IF nPlayerOne = 0 AND  nPlayerTwo = 0 THEN
	sWinner := '';
	xPlayerOneWins := FALSE;
	xPlayerTwoWins := FALSE;
END_IF

FOR i := 5 TO 49 DO //Set to 5 so as not to overwrite staff names

	IF 	CurrentMonthSignInTable[i].Name = '' THEN
	sPlayerList[i] := CurrentMonthSignInTable[i-5].Name;
	ELSE
	EXIT;	
	END_IF

END_FOR

ACTION Play11s:

END_ACTION

ACTION Play5s:

END_ACTION

END_PROGRAM

// ---- HMI/VariableHandleForHmi.TcPOU
PROGRAM VariableHandleForHmi
VAR
END_VAR

numberOfOpenWindows := EnOcean.totalNumberOfWindowsOpen;
boardroomModeIsProjector := LightControl.xBoardRoom_Lights_ProjectorMode;
boardroomModeIsFullOn := PTM200StrippedTables[3].Signal OR PTM200StrippedTables[2].Signal;
communalOccupancy1 := Dali.CommunalAreaPIR_1_Occupancy;
communalOccupancy2 := Dali.CommunalAreaPIR_2_Occupancy;
staffOccupancy1 := Dali.StaffroomPIR_1_Occupancy;
staffOccupancy2 := Dali.StaffroomPIR_2_Occupancy;
boardOccupancy1 := Dali.BoardroomPIR_1_Occupancy;
boardOccupancy2 := Dali.BoardroomPIR_2_Occupancy;
communalLux1 := Dali.CommunalAreaPIR_1_LuxLevel;
communalLux2 := Dali.CommunalAreaPIR_2_LuxLevel;
staffLux1 := Dali.StaffroomPIR_1_LuxLevel;
staffLux2 := Dali.StaffroomPIR_2_LuxLevel;
boardLux1 := Dali.BoardroomPIR_1_LuxLevel;
boardLux2 := Dali.BoardroomPIR_2_LuxLevel;

END_PROGRAM

// ---- WORKSHOP WALL/PowerSupply.TcPOU
PROGRAM PowerSupply
VAR
	triggerCoeRead							:	Pulse;
	readPsuDiagData							:	FB_EcCoESdoReadEx;
	readPsuInfoData							:	FB_EcCoESdoReadEx;
	psuDiagData								:	ST_PsuDiagData;
	psuInfoData								:	ST_PsuInfoData;
	testArr									:	ARRAY [1..20] OF BYTE;
	amsAdr							AT%I*	:	ST_AmsAddr;
	psuWarning						AT%I*	:	BOOL;
	psuError						AT%I*	:	BOOL;
	psuDcOk							AT%I*	:	BOOL;
	psuOutVoltage					AT%I*	:	REAL;
	psuOutCurrent					AT%I*	:	REAL;
	psuInputUnderVoltage			AT%I*	:	BOOL;
	psuDisableOutput				AT%Q*	:	BOOL;
END_VAR

triggerCoeRead(enable:= TRUE, offTime:= T#0.5S, onTime:= T#0.5S, Q=> );

readPsuDiagData(
	sNetId:= F_CreateAmsNetId(amsAdr.netId), 
	nSlaveAddr:= amsAdr.port, 
	nSubIndex:= 16#01, 
	nIndex:= 16#FA14, 
	pDstBuf:= ADR(psuDiagData), 
	cbBufLen:= SIZEOF(psuDiagData), 
	bExecute:= triggerCoeRead.Q, 
	tTimeout:= , 
	bCompleteAccess:= TRUE, 
	bBusy=> , 
	bError=> , 
	nErrId=> , 
	cbRead=> );
	
readPsuInfoData(
	sNetId:= F_CreateAmsNetId(amsAdr.netId), 
	nSlaveAddr:= amsAdr.port, 
	nSubIndex:= 16#01, 
	nIndex:= 16#F914, 
	pDstBuf:= ADR(psuInfoData), 
	cbBufLen:= SIZEOF(psuInfoData), 
	bExecute:= triggerCoeRead.Q, 
	tTimeout:= , 
	bCompleteAccess:= TRUE, 
	bBusy=> , 
	bError=> , 
	nErrId=> , 
	cbRead=> );

END_PROGRAM

// ---- BLINDS/ConvertBoolArrayToString.TcPOU
FUNCTION_BLOCK ConvertBoolArrayToString
VAR_INPUT
	boolArray: ARRAY[1..16] OF BOOL;
END_VAR
VAR_OUTPUT
	resultString: STRING := '';
END_VAR
VAR
	i: INT := 1;
END_VAR

FOR i := 1 TO 15 by 1 DO
    IF boolArray[i] THEN
        resultString := Concat(STR1 := resultString, STR2 := '1');
    ELSE
        resultString := Concat(STR1 := resultString, STR2 := '0');
    END_IF;
END_FOR;

END_FUNCTION_BLOCK

// ---- BLINDS/fConvertBoolArrayToString.TcPOU
FUNCTION fConvertBoolArrayToString : STRING
VAR_INPUT
	boolArray: ARRAY[1..16] OF BOOL;
END_VAR
VAR
	i: INT := 1;
END_VAR

FOR i := 1 TO 16 BY 1 DO
    IF boolArray[i] THEN
        fConvertBoolArrayToString := Concat(STR1 := fConvertBoolArrayToString, STR2 := '1');
    ELSE
        fConvertBoolArrayToString := Concat(STR1 := fConvertBoolArrayToString, STR2 := '0');
    END_IF;
END_FOR;

END_FUNCTION

// ---- BLINDS/PrgMqttCom_Blinds_Publisher.TcPOU
PROGRAM PrgMqttCom_Blinds_Publisher
VAR
	fbMqttClient : FB_IotMqttClient;
	bSetParameter : BOOL := TRUE;
	bConnect : BOOL := TRUE;
	
	(* published message *)
	sTopicSelectRoom : STRING(255);//:= 'Staff Room';
	sTopicSelectBulkCommand : STRING(255) := 'Blind Selection';
	//sTopicSelectBoardroom : STRING(255) := 'Boardroom';
	
	bSelectStaffRoom : BOOL;
	bSelectCommunalArea : BOOL;
	bSelectBoardroom : BOOL;
	
	sPayloadCommand : STRING(255);// := 'Up';
//	sPayloadCommandDown : STRING(255) := 'Down';
//	sPayloadCommandStop : STRING(255) := 'Stop';
//	sPayloadCommandTilt : STRING(255) := 'Tilt';

	bCommandUp : BOOL;
	bCommandDown : BOOL;
	bCommandStop : BOOL;
	bCommandTilt : BOOL;
	
	bulkCommandPackage :STRING;
	
	i: INT;
	fbTimer : TON := (PT:=T#1S);
	fbTimerTilt : TON := (PT:=T#0.5S);
	
	fbMessageQueue : FB_IotMqttMessageQueue;
	fbMessage : FB_IotMqttMessage;
	
	hrErrorOccurred : HRESULT; // contains the latest occurred error
END_VAR

IF bSetParameter THEN
	bSetParameter := FALSE;
	fbMqttClient.sHostName:= '10.199.143.2';
	fbMqttClient.nHostPort:= 1883;
	fbMqttClient.sClientId:= 'CX2040_Blinds'; 
	fbMqttClient.sTopicPrefix:= ''; 
	fbMqttClient.nKeepAlive:= 60; 
//	fbMqttClient.sUserName:= ;
//	fbMqttClient.sUserPassword:= ; 
//	fbMqttClient.stWill:= ; 
//	fbMqttClient.stTLS:= ;
	fbMqttClient.ipMessageQueue := fbMessageQueue;
END_IF

fbMqttClient.Execute(bConnect);
IF fbMqttClient.bError THEN
	// add your error logging here
	hrErrorOccurred := fbMqttClient.hrErrorCode;
END_IF

IF bSelectStaffRoom THEN
	bSelectStaffRoom := FALSE;
	sTopicSelectRoom := 'Staff Room';
	bulkCommandPackage := fConvertBoolArrayToString(boolArray := BackgroundComms.BlindCommandTable[0].SelectBlindsBulkCommand);
END_IF

IF bSelectCommunalArea THEN
	bSelectCommunalArea := FALSE;
	sTopicSelectRoom := 'Communal Area';
	bulkCommandPackage := fConvertBoolArrayToString(boolArray := BackgroundComms.BlindCommandTable[1].SelectBlindsBulkCommand);
END_IF

IF bSelectBoardroom THEN
	bSelectBoardroom := FALSE;
	sTopicSelectRoom := 'Boardroom';
	bulkCommandPackage := fConvertBoolArrayToString(boolArray := BackgroundComms.BlindCommandTable[2].SelectBlindsBulkCommand);
END_IF



IF bCommandUp THEN
	bCommandUp := FALSE;
	sPayloadCommand := 'Up';
	IF sTopicSelectRoom = 'Staff Room' THEN
		bSelectStaffRoom := TRUE;
	ELSIF sTopicSelectRoom = 'Communal Area' THEN
		bulkCommandPackage := fConvertBoolArrayToString(boolArray := BackgroundComms.BlindCommandTable[1].SelectBlindsBulkCommand);
	ELSIF sTopicSelectRoom = 'Boardroom' THEN
		bulkCommandPackage := fConvertBoolArrayToString(boolArray := BackgroundComms.BlindCommandTable[2].SelectBlindsBulkCommand);
	END_IF
END_IF

IF bCommandDown THEN
	bCommandDown := FALSE;
	sPayloadCommand := 'Down';
	IF sTopicSelectRoom = 'Staff Room' THEN
		bSelectStaffRoom := TRUE;//bulkCommandPackage := fConvertBoolArrayToString(boolArray := BackgroundComms.BlindCommandTable[0].SelectBlindsBulkCommand);
	ELSIF sTopicSelectRoom = 'Communal Area' THEN
		bulkCommandPackage := fConvertBoolArrayToString(boolArray := BackgroundComms.BlindCommandTable[1].SelectBlindsBulkCommand);
	ELSIF sTopicSelectRoom = 'Boardroom' THEN
		bulkCommandPackage := fConvertBoolArrayToString(boolArray := BackgroundComms.BlindCommandTable[2].SelectBlindsBulkCommand);
	END_IF
END_IF

IF bCommandStop THEN
	bCommandStop := FALSE;
	sPayloadCommand := 'Stop';
	IF sTopicSelectRoom = 'Staff Room' THEN
		bSelectStaffRoom := TRUE;//bulkCommandPackage := fConvertBoolArrayToString(boolArray := BackgroundComms.BlindCommandTable[0].SelectBlindsBulkCommand);
	ELSIF sTopicSelectRoom = 'Communal Area' THEN
		bulkCommandPackage := fConvertBoolArrayToString(boolArray := BackgroundComms.BlindCommandTable[1].SelectBlindsBulkCommand);
	ELSIF sTopicSelectRoom = 'Boardroom' THEN
		bulkCommandPackage := fConvertBoolArrayToString(boolArray := BackgroundComms.BlindCommandTable[2].SelectBlindsBulkCommand);
	END_IF
END_IF

IF bCommandTilt THEN
	bCommandTilt := FALSE;
	sPayloadCommand := 'Tilt';
	IF sTopicSelectRoom = 'Staff Room' THEN
		bSelectStaffRoom := TRUE;//bulkCommandPackage := fConvertBoolArrayToString(boolArray := BackgroundComms.BlindCommandTable[0].SelectBlindsBulkCommand);
	ELSIF sTopicSelectRoom = 'Communal Area' THEN
		bulkCommandPackage := fConvertBoolArrayToString(boolArray := BackgroundComms.BlindCommandTable[1].SelectBlindsBulkCommand);
	ELSIF sTopicSelectRoom = 'Boardroom' THEN
		bulkCommandPackage := fConvertBoolArrayToString(boolArray := BackgroundComms.BlindCommandTable[2].SelectBlindsBulkCommand);
	END_IF
END_IF





IF fbMqttClient.bConnected THEN
	IF sPayloadCommand = 'Tilt' THEN
		fbTimerTilt(IN:=TRUE);
		fbMqttClient.Publish(	sTopic:= sTopicSelectBulkCommand, 
									pPayload:= ADR(bulkCommandPackage), nPayloadSize:= LEN2(ADR(bulkCommandPackage))+1, 
									eQoS:= TcIotMqttQos.AtMostOnceDelivery, bRetain:= FALSE, bQueue:= FALSE );
		fbMqttClient.Publish(	sTopic:= sTopicSelectRoom, 
									pPayload:= ADR(sPayloadCommand), nPayloadSize:= LEN2(ADR(sPayloadCommand))+1, 
									eQoS:= TcIotMqttQos.AtMostOnceDelivery, bRetain:= FALSE, bQueue:= FALSE );
		
		IF fbTimerTilt.Q THEN // publish new payload every second
			sPayloadCommand := 'Stop';
			fbTimerTilt(IN:=FALSE);
			fbMqttClient.Publish(	sTopic:= sTopicSelectBulkCommand, 
									pPayload:= ADR(bulkCommandPackage), nPayloadSize:= LEN2(ADR(bulkCommandPackage))+1, 
									eQoS:= TcIotMqttQos.AtMostOnceDelivery, bRetain:= FALSE, bQueue:= FALSE );
			fbMqttClient.Publish(	sTopic:= sTopicSelectRoom, 
									pPayload:= ADR(sPayloadCommand), nPayloadSize:= LEN2(ADR(sPayloadCommand))+1, 
									eQoS:= TcIotMqttQos.AtMostOnceDelivery, bRetain:= FALSE, bQueue:= FALSE );			
			IF fbMqttClient.bError THEN
				// add your error logging here
				hrErrorOccurred := fbMqttClient.hrErrorCode;
			END_IF
		END_IF
	ELSE
		fbTimer(IN:=TRUE);
		IF fbTimer.Q THEN // publish new payload every second
			fbTimer(IN:=FALSE);
			fbMqttClient.Publish(	sTopic:= sTopicSelectBulkCommand, 
									pPayload:= ADR(bulkCommandPackage), nPayloadSize:= LEN2(ADR(bulkCommandPackage))+1, 
									eQoS:= TcIotMqttQos.AtMostOnceDelivery, bRetain:= FALSE, bQueue:= FALSE );
									
			fbMqttClient.Publish(	sTopic:= sTopicSelectRoom, 
									pPayload:= ADR(sPayloadCommand), nPayloadSize:= LEN2(ADR(sPayloadCommand))+1, 
									eQoS:= TcIotMqttQos.AtMostOnceDelivery, bRetain:= FALSE, bQueue:= FALSE );
			IF fbMqttClient.bError THEN
				// add your error logging here
				hrErrorOccurred := fbMqttClient.hrErrorCode;
			END_IF
		END_IF
	END_IF
END_IF

fbTimerTilt();

END_PROGRAM

// ---- HMI/ReadCP67.TcPOU
PROGRAM ReadCP67
VAR
	
	ReadActLightLvlBoardroom :FB_DALIV2QueryActualLevel;  //Used to read back actual light lvl to correct dimmer on CP67 ask Plug top


	ADS_READ:ADSREAD;
	
	ADX_READ_DMXR:ADSREAD;
	ADX_READ_DMXG:ADSREAD;
	ADX_READ_DMXB:ADSREAD;
	
	DMX_Enable_READ:ADSREAD;
	
	HoldCP67BoardRoomLightsOn:BYTE;
	

	Sample		: BYTE;
	
	DMXRValues	:	ARRAY [0..7] OF BYTE;
	DMXGValues	:	ARRAY [0..7] OF BYTE;
	DMXBValues	:	ARRAY [0..7] OF BYTE;
	
	CP67_DMX_Enable	:	BOOL;
	
	FBDALIV2Dimmer1Switch : ARRAY [1..15] OF FB_DALIV2Dimmer1Switch;
	CASECP67BoardRoomLightsOn : INT;

END_VAR

sample := sample + 1;

FBDALIV2Dimmer1Switch[1](stCommandBuffer:= stCommandBuffer);
FBDALIV2Dimmer1Switch[2](stCommandBuffer:= stCommandBuffer);
ReadActLightLvlBoardroom(stCommandBuffer := stCommandBuffer , nActualLevel => BoardroomActualLightLvl ); 

IF CP67BoardRoomLightsOn <> HoldCP67BoardRoomLightsOn THEN
HoldCP67BoardRoomLightsOn := CP67BoardRoomLightsOn;
CASECP67BoardRoomLightsOn := 10;
END_IF

	CASE CASECP67BoardRoomLightsOn OF
		
	0: //Idle
	
	10:	FBDALIV2Dimmer1Switch[1].nDimmValue	:=  CP67BoardRoomLightsOn;
		FBDALIV2Dimmer1Switch[1].nAddr		:= 3;
		FBDALIV2Dimmer1Switch[1].eAddrType	:= 1;
			
		FBDALIV2Dimmer1Switch[2].nDimmValue	:=  CP67BoardRoomLightsOn; 
		FBDALIV2Dimmer1Switch[2].nAddr		:= 2; 
		FBDALIV2Dimmer1Switch[2].eAddrType	:= 1;
			
		CASECP67BoardRoomLightsOn			:= 20;	
			
	20:	IF  NOT FBDALIV2Dimmer1Switch[1].bBusy AND NOT FBDALIV2Dimmer1Switch[2].bBusy THEN
		CASECP67BoardRoomLightsOn 			:= 30;	

		ReadActLightLvlBoardroom.bStart		:= TRUE;
		ReadActLightLvlBoardroom.nAddr		:= 6;
		ReadActLightLvlBoardroom.eAddrType	:= 0;
		END_IF
	
	30:	IF NOT ReadActLightLvlBoardroom.bBusy THEN
		ReadActLightLvlBoardroom.bStart			:= FALSE;
		CASECP67BoardRoomLightsOn 				:= 0;
		
		END_IF
				
		
	END_CASE
		
	
	
	
(*// Send back actual light lvls for slider on CP67	
ReadActLightLvlBoardroom(
	bStart:= Sample.0, 
	nAddr:= 6, 
	eAddrType:= 0, 
	eCommandPriority:= , 
	bBusy=> , 
	bError=> , 
	nErrorId=> , 
	nActualLevel=> BoardroomActualLightLvl, 
	stCommandBuffer:= stCommandBuffer);	*)

(*
// DMX Values	
ADX_READ_DMXR(
	NETID:= '192.168.3.8.1.1', 
	PORT:= 851, 
	IDXGRP:= 16#4020, 
	IDXOFFS:= 1, 
	LEN:= 8, 
	DESTADDR:= ADR(DMXRValues), 
	READ:= Sample.0, 
	TMOUT:= T#2S, 
	BUSY=> , 
	ERR=> , 
	ERRID=> );
	
ADX_READ_DMXG(
	NETID:= '192.168.3.8.1.1', 
	PORT:= 851, 
	IDXGRP:= 16#4020, 
	IDXOFFS:= 9, 
	LEN:= 8, 
	DESTADDR:= ADR(DMXGValues), 
	READ:= Sample.0, 
	TMOUT:= T#2S, 
	BUSY=> , 
	ERR=> , 
	ERRID=> );
	
ADX_READ_DMXB(
	NETID:= '192.168.3.8.1.1', 
	PORT:= 851, 
	IDXGRP:= 16#4020, 
	IDXOFFS:= 17, 
	LEN:= 8, 
	DESTADDR:= ADR(DMXBValues), 
	READ:= Sample.0, 
	TMOUT:= T#2S, 
	BUSY=> , 
	ERR=> , 
	ERRID=> );
	
	
DMX_Enable_READ(
	NETID:= '192.168.3.8.1.1', 
	PORT:= 851, 
	IDXGRP:= 16#4020, 
	IDXOFFS:= 25, 
	LEN:= 1, 
	DESTADDR:= ADR(CP67_DMX_Enable), 
	READ:= Sample.0, 
	TMOUT:= T#2S, 
	BUSY=> , 
	ERR=> , 
	ERRID=> );
	*)

END_PROGRAM

// ---- ML/FB_CoffeeFifo.TcPOU
FUNCTION_BLOCK FB_CoffeeFifo
VAR_INPUT
	bOverwrite	: BOOL;
	in 			: REAL;
END_VAR
VAR_OUTPUT
	bOk			: BOOL;
	nCount		: UDINT;
	nLoad		: UDINT;
	out			: REAL;
	arrBuffer 	: ARRAY[0..MAX_BUFFER_SIZE] OF LREAL; (* Buffer memory used by FB_MemRingBuffer function block *)
END_VAR
VAR
	//arrBuffer 	: ARRAY[0..MAX_BUFFER_SIZE] OF lREAL; (* Buffer memory used by FB_MemRingBuffer function block *)
	fbBuffer	: FB_MemRingBuffer;
END_VAR

VAR CONSTANT
    MAX_BUFFER_SIZE : UDINT := 160;
END_VAR

ACTION A_Add:
fbBuffer.A_AddTail( pWrite:= ADR( in ),
					cbWrite:= SIZEOF( in ),
					pBuffer:= ADR( arrBuffer ),
					cbBuffer:= SIZEOF( arrBuffer ),
					bOk=> bOk,
					nCount => nCount );


IF NOT bOk THEN (* overflow ? *)
	IF bOverwrite THEN
		fbBuffer.A_RemoveHead(); (* remove one oldest entry *)
		
		fbBuffer.A_AddTail( bOk => bOk, nCount => nCount );
	END_IF
END_IF



nLoad := (fbBuffer.cbSize * 100) / MAX_BUFFER_SIZE;
END_ACTION

ACTION A_Get:
fbBuffer.A_GetHead( pRead:= ADR( out ),
					cbRead:= SIZEOF( out ),
					pBuffer:= ADR( arrBuffer ),
					cbBuffer:= SIZEOF( arrBuffer ),
					bOk=> bOk,
					nCount => nCount );

nLoad := (fbBuffer.cbSize * 100) / MAX_BUFFER_SIZE;;
END_ACTION

ACTION A_Remove:
fbBuffer.A_RemoveHead( 	pRead:= ADR( out ),
						cbRead:= SIZEOF( out ),
						pBuffer:= ADR( arrBuffer ),
						cbBuffer:= SIZEOF( arrBuffer ),
						bOk=> bOk,
						nCount => nCount );

nLoad := (fbBuffer.cbSize * 100) / MAX_BUFFER_SIZE;
END_ACTION

ACTION A_Reset:
MEMSET( ADR( arrBuffer ), 0, SIZEOF( arrBuffer ) ); (* reset (optional) internal buffer *)

fbBuffer.A_Reset( 	bOk=> bOk,
					nCount => nCount );

nLoad := (fbBuffer.cbSize * 100) / MAX_BUFFER_SIZE;
END_ACTION

END_FUNCTION_BLOCK
